// TIA Portal V20 export
// export: Created 2025-12-01T14:56:14.430751Z, ExportSetting None, DisplayName Totally Integrated Automation Portal, DisplayVersion V20 Update 3, DisplayName TIA Portal Openness, DisplayVersion V20 Update 3, DisplayName TIA Portal Version Control Interface, DisplayVersion V20 Update 3, DisplayName STEP 7 Professional, DisplayVersion V20 Update 3, DisplayName STEP 7 Safety, DisplayVersion V20 Update 2, DisplayName WinCC Basic/Comfort/Advanced, DisplayVersion V20 Update 3, DisplayName WinCC Professional, DisplayVersion V20 Update 3, DisplayName WinCC Unified, DisplayVersion V20 Update 3
TYPE "UDT_ProtocoloRecDispositivo"
   STRUCT
      Bit_00 : Bool;
      Error : Bool;   // Orden de Error del JdT
      Rearme : Bool;   // Orden de Rearme
      ParoBlando : Bool;   // Orden de Paro Blando
      Reset : Bool;   // Orden de Reset
      Paro : Bool;   // Orden de Paro
      Marcha : Bool;   // Orden de Marcha
      Bit_07 : Bool;
      Automatico : Bool;   // Orden de Automatico
      Manual : Bool;   // Orden de Manual
      Mantenimiento : Bool;
      Bit_13 : Bool;
      Bit_14 : Bool;
      Bit_15 : Bool;
      Bit_16 : Bool;
      EmiOK : Bool;   // Emision OK de la Presencia
   END_STRUCT;
END_TYPE
